INTERFACE I_Middleware

METHOD Handle
VAR_INPUT
	Request : I_Request;
	Response : I_ServerResponse;
END_VAR
END_METHOD

PROPERTY PUBLIC NextMiddleware : I_Middleware
GET
END_GET
SET
END_SET
END_PROPERTY

END_INTERFACE

(* stored: Version 1.1.0.1, ProductVersion 3.1.4024.12
   Itf I_Middleware: Id {51943325-82a1-0ea1-047d-2b679976e290}
   Method Handle: Id {7ea728ba-e48a-031a-006d-0f4a9380f152}
   Property NextMiddleware: Id {4390db13-72e0-0493-1d74-493592b31b1f}
   Get Get: Id {53bfdbde-4ca7-0f73-1199-758d164509f6}
   Set Set: Id {e4bf52c1-31ce-075e-2e7d-be8114cc80f7} *)
